(*

.. <legal notes>

legal notes
=================
| SPDX-FileCopyrightText: © 2026 Oleksandr Tiutyk <trofimich@gmail.com>
| SPDX-License-Identifier: LGPL-3.0-only
| For details check: LGPL-3.0-only_

.. _LGPL-3.0-only: https://www.gnu.org/licenses/lgpl-3.0.en.html

.. </legal notes>

*)

FUNCTION_BLOCK ABSTRACT SimpleDevice EXTENDS Device IMPLEMENTS ISimpleDevice

{attribute 'monitoring' := 'call'}
PROPERTY ABSTRACT BoundToIO : BOOL
GET
END_GET
END_PROPERTY

METHOD FINAL Disable
IF NOT _Enabled THEN
	RETURN;
END_IF

OnEnabledChange(FALSE);

_Enabled := FALSE;
END_METHOD

METHOD FINAL Enable
VAR_INPUT
	includeChildren : BOOL := TRUE;
END_VAR
IF BoundToIO THEN
	RETURN;
END_IF

OnEnabledChange(TRUE);

_Enabled := TRUE;

Parent.Enable(FALSE);
END_METHOD

METHOD FINAL Initialize : BOOL
VAR
	memberNotSpecifiedException : Core.DataMemberNotSpecifiedException;	
END_VAR
IF _Parent = 0 THEN
	memberNotSpecifiedException.Throw(Namespacename, ClassName, __POUNAME(), __POSITION(), 'Parent');
END_IF

Initialize := OnInitialize();
END_METHOD

METHOD PROTECTED OnEnabledChange 
VAR_INPUT
	newValue : BOOL;
END_VAR
END_METHOD

METHOD PROTECTED OnInitialize : BOOL
OnInitialize := TRUE;
END_METHOD

END_FUNCTION_BLOCK

(* stored: Version 1.1.0.1
   POU SimpleDevice: Id {7c21300f-1ad4-4217-9d49-d0f060249ecb}, SpecialFunc None
   Folder Internal members to override: Id {78a2b14c-f3bd-4833-8b88-abed9d422e8c}
   Property BoundToIO: Id {b628aa04-eeeb-4d72-affe-9ddf01c0664c}
   Get Get: Id {5d4063e8-5bcc-4414-818d-9d72aff3da84}
   Method Disable: Id {456e8034-80c7-4023-bbc1-b1fa7ea41430}
   Method Enable: Id {da30d30f-9904-4df0-aa77-06867eb85fe2}
   Method Initialize: Id {b3b19006-a5ea-4fbb-ad1a-6167b8192dbd}
   Method OnEnabledChange: Id {1850d5ad-feab-4558-b561-a14df8e5fb12}
   Method OnInitialize: Id {896e6103-6f85-4d68-a85e-f1c9cefc8e44} *)
